TYPE VelocityCtrl_Error_typ :
	STRUCT
		ErrorID : UDINT ;
		ErrorText : STRING[2048];(*ARRAY[0..3]OF STRING[79]*) (*Error Text*)
		ErrorEntry: Eh_ErrorEntry_typ;
	END_STRUCT
END_TYPE

(* stored: Version 1.1.0.1, ProductVersion 3.1.4024.3
   DUT VelocityCtrl_Error_typ: Id {e29514cc-bcd1-4604-b026-7e6cca564b81} *)
